KUKA KRL program: test.src

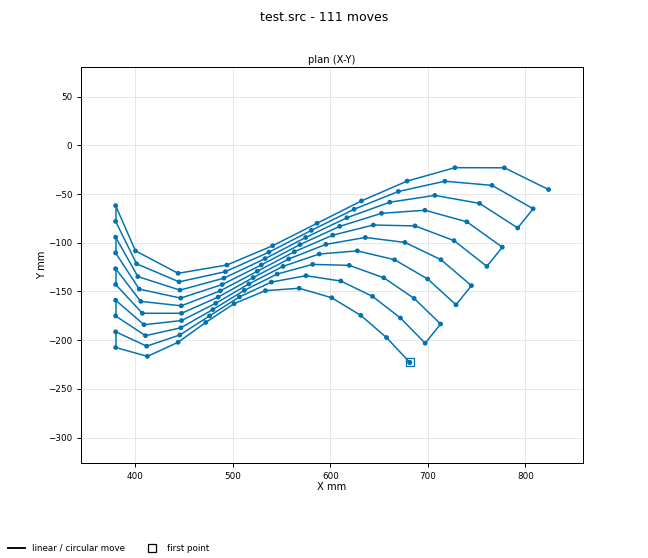
[picture p0: tool path of test.src, 111 of 113 moves have a stored position in this frame; points joined in program order, loops and branches not executed]
&ACCESS RVP
&REL 1
&PARAM TEMPLATE = C:\KRC\Roboter\Template\vorgabe
&PARAM EDITMASK = *
DEF test ( )


;FOLD INI
;FOLD BASISTECH INI
GLOBAL INTERRUPT DECL 3 WHEN $STOPMESS==TRUE DO IR_STOPM ( )
INTERRUPT ON 3
BAS (#INITMOV,0 )
;ENDFOLD (BASISTECH INI)
;ENDFOLD (INI)

;FOLD STARTPOSITION - BASE IS 0, TOOL IS 0, SPEED IS 15%, POSITION IS A1 5,A2 -90,A3 100,A4 5,A5 10,A6 -5,E1 0,E2 0,E3 0,E4 0
$BWDSTART = FALSE
PDAT_ACT = {VEL 15,ACC 100,APO_DIST 50}
FDAT_ACT = {TOOL_NO 0,BASE_NO 0,IPO_FRAME #BASE}
BAS (#PTP_PARAMS,15)
PTP  {A1 5,A2 -90,A3 100,A4 5,A5 10,A6 -5,E1 0,E2 0,E3 0,E4 0}
;ENDFOLD

;FOLD LIN SPEED IS 0.25 m/sec, INTERPOLATION SETTINGS IN FOLD
$VEL.CP=0.25
$APO.CDIS=10
$ADVANCE=3
;ENDFOLD

$OUT_C[1]=TRUE
PTP {E6POS: X 681.378, Y -222.764, Z 500, A 0, B -90, C 40.701, E1 0, E2 0, E3 0, E4 0, S 'B 110'} C_PTP
$VEL.CP=0.11208624
$OUT_C[1]=TRUE
LIN {E6POS: X 681.378, Y -222.764, Z 500, A 0, B -90, C 40.701, E1 0, E2 0, E3 0, E4 0} C_DIS
$VEL.CP=0.1175562
LIN {E6POS: X 657.556, Y -197.262, Z 500, A 0, B -90, C 45.729, E1 0, E2 0, E3 0, E4 0} C_DIS
$VEL.CP=0.12712281
LIN {E6POS: X 631.136, Y -174.483, Z 500, A 0, B -90, C 53.29, E1 0, E2 0, E3 0, E4 0} C_DIS
$VEL.CP=0.14338495
LIN {E6POS: X 601.341, Y -156.414, Z 500, A 0, B -90, C 65.177, E1 0, E2 0, E3 0, E4 0} C_DIS
$VEL.CP=0.16124801
LIN {E6POS: X 567.97, Y -146.683, Z 500, A 0, B -90, C 83.337, E1 0, E2 0, E3 0, E4 0} C_DIS
$VEL.CP=0.15591648
LIN {E6POS: X 533.344, Y -149.111, Z 500, A 0, B -90, C 104.356, E1 0, E2 0, E3 0, E4 0} C_DIS
$VEL.CP=0.13138869
LIN {E6POS: X 501.213, Y -162.493, Z 500, A 0, B -90, C 119.461, E1 0, E2 0, E3 0, E4 0} C_DIS
$VEL.CP=0.10713721
LIN {E6POS: X 472.106, Y -181.729, Z 500, A 0, B -90, C 126.091, E1 0, E2 0, E3 0, E4 0} C_DIS
$VEL.CP=0.12689649
LIN {E6POS: X 443.773, Y -202.115, Z 500, A 0, B -90, C 123.452, E1 0, E2 0, E3 0, E4 0} C_DIS
$VEL.CP=0.22954467
LIN {E6POS: X 412.246, Y -216.53, Z 500, A 0, B -90, C 99.792, E1 0, E2 0, E3 0, E4 0} C_DIS
$VEL.CP=0.19782427
LIN {E6POS: X 379.699, Y -207.447, Z 500, A 0, B -90, C 51.492, E1 0, E2 0, E3 0, E4 0} C_DIS
$VEL.CP=0.18350544
LIN {E6POS: X 379.699, Y -191.28, Z 500, A 0, B -90, C -136.662, E1 0, E2 0, E3 0, E4 0} C_DIS
$VEL.CP=0.242284
LIN {E6POS: X 411.548, Y -206.08, Z 500, A 0, B -90, C -88.625, E1 0, E2 0, E3 0, E4 0} C_DIS
$VEL.CP=0.13252691
LIN {E6POS: X 445.551, Y -194.567, Z 500, A 0, B -90, C -60.589, E1 0, E2 0, E3 0, E4 0} C_DIS
$VEL.CP=0.10130669
LIN {E6POS: X 476.069, Y -175.016, Z 500, A 0, B -90, C -56.087, E1 0, E2 0, E3 0, E4 0} C_DIS
$VEL.CP=0.12101501
LIN {E6POS: X 506.648, Y -155.559, Z 500, A 0, B -90, C -60.177, E1 0, E2 0, E3 0, E4 0} C_DIS
$VEL.CP=0.14114481
LIN {E6POS: X 539.479, Y -140.317, Z 500, A 0, B -90, C -71.221, E1 0, E2 0, E3 0, E4 0} C_DIS
$VEL.CP=0.15549513
LIN {E6POS: X 574.997, Y -133.814, Z 500, A 0, B -90, C -88.912, E1 0, E2 0, E3 0, E4 0} C_DIS
$VEL.CP=0.14877746
LIN {E6POS: X 610.665, Y -139.264, Z 500, A 0, B -90, C -108.055, E1 0, E2 0, E3 0, E4 0} C_DIS
$VEL.CP=0.13304864
LIN {E6POS: X 643.215, Y -155.004, Z 500, A 0, B -90, C -122.625, E1 0, E2 0, E3 0, E4 0} C_DIS
$VEL.CP=0.1215327
LIN {E6POS: X 671.847, Y -177.173, Z 500, A 0, B -90, C -132.204, E1 0, E2 0, E3 0, E4 0} C_DIS
$VEL.CP=0.11461978
LIN {E6POS: X 697.2, Y -203.06, Z 500, A 0, B -90, C -138.566, E1 0, E2 0, E3 0, E4 0} C_DIS
$VEL.CP=0.11747553
LIN {E6POS: X 713.022, Y -183.357, Z 500, A 0, B -90, C 42.204, E1 0, E2 0, E3 0, E4 0} C_DIS
$VEL.CP=0.12604367
LIN {E6POS: X 685.918, Y -157.123, Z 500, A 0, B -90, C 50.194, E1 0, E2 0, E3 0, E4 0} C_DIS
$VEL.CP=0.13895214
LIN {E6POS: X 654.762, Y -135.927, Z 500, A 0, B -90, C 62.153, E1 0, E2 0, E3 0, E4 0} C_DIS
$VEL.CP=0.15060037
LIN {E6POS: X 619.368, Y -123.2, Z 500, A 0, B -90, C 79.05, E1 0, E2 0, E3 0, E4 0} C_DIS
$VEL.CP=0.14631891
LIN {E6POS: X 581.798, Y -122.186, Z 500, A 0, B -90, C 97.587, E1 0, E2 0, E3 0, E4 0} C_DIS
$VEL.CP=0.12977299
LIN {E6POS: X 545.471, Y -132.089, Z 500, A 0, B -90, C 111.844, E1 0, E2 0, E3 0, E4 0} C_DIS
$VEL.CP=0.11350675
LIN {E6POS: X 511.672, Y -148.834, Z 500, A 0, B -90, C 119.873, E1 0, E2 0, E3 0, E4 0} C_DIS
$VEL.CP=0.1031691
LIN {E6POS: X 479.457, Y -168.509, Z 500, A 0, B -90, C 121.926, E1 0, E2 0, E3 0, E4 0} C_DIS
$VEL.CP=0.13868728
LIN {E6POS: X 446.677, Y -187.191, Z 500, A 0, B -90, C 115.335, E1 0, E2 0, E3 0, E4 0} C_DIS
$VEL.CP=0.24988499
LIN {E6POS: X 410.331, Y -195.313, Z 500, A 0, B -90, C 82.591, E1 0, E2 0, E3 0, E4 0} C_DIS
$VEL.CP=0.17049267
LIN {E6POS: X 379.699, Y -175.112, Z 500, A 0, B -90, C 36.664, E1 0, E2 0, E3 0, E4 0} C_DIS
$VEL.CP=0.15965107
LIN {E6POS: X 379.699, Y -158.945, Z 500, A 0, B -90, C -148.742, E1 0, E2 0, E3 0, E4 0} C_DIS
$VEL.CP=0.25
LIN {E6POS: X 408.793, Y -184.08, Z 500, A 0, B -90, C -106.079, E1 0, E2 0, E3 0, E4 0} C_DIS
$VEL.CP=0.14513617
LIN {E6POS: X 447.236, Y -179.828, Z 500, A 0, B -90, C -68.773, E1 0, E2 0, E3 0, E4 0} C_DIS
$VEL.CP=0.10734447
LIN {E6POS: X 482.361, Y -162.109, Z 500, A 0, B -90, C -60.049, E1 0, E2 0, E3 0, E4 0} C_DIS
$VEL.CP=0.10792353
LIN {E6POS: X 516.364, Y -142.247, Z 500, A 0, B -90, C -60.383, E1 0, E2 0, E3 0, E4 0} C_DIS
$VEL.CP=0.12129846
LIN {E6POS: X 551.369, Y -124.246, Z 500, A 0, B -90, C -66.049, E1 0, E2 0, E3 0, E4 0} C_DIS
$VEL.CP=0.13674186
LIN {E6POS: X 588.577, Y -111.545, Z 500, A 0, B -90, C -77.229, E1 0, E2 0, E3 0, E4 0} C_DIS
$VEL.CP=0.14833769
LIN {E6POS: X 627.681, Y -108.322, Z 500, A 0, B -90, C -94.073, E1 0, E2 0, E3 0, E4 0} C_DIS
$VEL.CP=0.14398834
LIN {E6POS: X 665.817, Y -117.427, Z 500, A 0, B -90, C -112.461, E1 0, E2 0, E3 0, E4 0} C_DIS
$VEL.CP=0.13105502
LIN {E6POS: X 699.766, Y -137.17, Z 500, A 0, B -90, C -127.03, E1 0, E2 0, E3 0, E4 0} C_DIS
$VEL.CP=0.12069929
LIN {E6POS: X 728.844, Y -163.654, Z 500, A 0, B -90, C -136.944, E1 0, E2 0, E3 0, E4 0} C_DIS
$VEL.CP=0.1243438
LIN {E6POS: X 744.665, Y -143.95, Z 500, A 0, B -90, C 43.947, E1 0, E2 0, E3 0, E4 0} C_DIS
$VEL.CP=0.13643728
LIN {E6POS: X 713.389, Y -117.376, Z 500, A 0, B -90, C 56.167, E1 0, E2 0, E3 0, E4 0} C_DIS
$VEL.CP=0.14714289
LIN {E6POS: X 676.456, Y -99.656, Z 500, A 0, B -90, C 73.323, E1 0, E2 0, E3 0, E4 0} C_DIS
$VEL.CP=0.14302107
LIN {E6POS: X 635.84, Y -94.578, Z 500, A 0, B -90, C 92.121, E1 0, E2 0, E3 0, E4 0} C_DIS
$VEL.CP=0.12834552
LIN {E6POS: X 595.443, Y -101.629, Z 500, A 0, B -90, C 106.677, E1 0, E2 0, E3 0, E4 0} C_DIS
$VEL.CP=0.11500083
LIN {E6POS: X 557.21, Y -116.656, Z 500, A 0, B -90, C 115.335, E1 0, E2 0, E3 0, E4 0} C_DIS
$VEL.CP=0.10366841
LIN {E6POS: X 520.795, Y -135.736, Z 500, A 0, B -90, C 119.205, E1 0, E2 0, E3 0, E4 0} C_DIS
$VEL.CP=0.11093951
LIN {E6POS: X 484.87, Y -155.738, Z 500, A 0, B -90, C 118.025, E1 0, E2 0, E3 0, E4 0} C_DIS
$VEL.CP=0.15165687
LIN {E6POS: X 447.326, Y -172.357, Z 500, A 0, B -90, C 107.094, E1 0, E2 0, E3 0, E4 0} C_DIS
$VEL.CP=0.24285384
LIN {E6POS: X 407.124, Y -172.341, Z 500, A 0, B -90, C 65.741, E1 0, E2 0, E3 0, E4 0} C_DIS
$VEL.CP=0.15093802
LIN {E6POS: X 379.699, Y -142.777, Z 500, A 0, B -90, C 26.821, E1 0, E2 0, E3 0, E4 0} C_DIS
$VEL.CP=0.14400658
LIN {E6POS: X 379.699, Y -126.61, Z 500, A 0, B -90, C -156.794, E1 0, E2 0, E3 0, E4 0} C_DIS
$VEL.CP=0.23087273
LIN {E6POS: X 405.466, Y -160.137, Z 500, A 0, B -90, C -121.592, E1 0, E2 0, E3 0, E4 0} C_DIS
$VEL.CP=0.15801723
LIN {E6POS: X 447.042, Y -164.693, Z 500, A 0, B -90, C -77.117, E1 0, E2 0, E3 0, E4 0} C_DIS
$VEL.CP=0.11407162
LIN {E6POS: X 487.06, Y -149.339, Z 500, A 0, B -90, C -63.896, E1 0, E2 0, E3 0, E4 0} C_DIS
$VEL.CP=0.10035442
LIN {E6POS: X 525.025, Y -129.253, Z 500, A 0, B -90, C -61.385, E1 0, E2 0, E3 0, E4 0} C_DIS
$VEL.CP=0.1102753
LIN {E6POS: X 563.021, Y -109.226, Z 500, A 0, B -90, C -63.717, E1 0, E2 0, E3 0, E4 0} C_DIS
$VEL.CP=0.12153792
LIN {E6POS: X 602.44, Y -92.222, Z 500, A 0, B -90, C -70.369, E1 0, E2 0, E3 0, E4 0} C_DIS
$VEL.CP=0.136359
LIN {E6POS: X 644.03, Y -81.81, Z 500, A 0, B -90, C -82.534, E1 0, E2 0, E3 0, E4 0} C_DIS
$VEL.CP=0.14766606
LIN {E6POS: X 686.794, Y -82.719, Z 500, A 0, B -90, C -100.715, E1 0, E2 0, E3 0, E4 0} C_DIS
$VEL.CP=0.14192006
LIN {E6POS: X 726.787, Y -97.808, Z 500, A 0, B -90, C -120.207, E1 0, E2 0, E3 0, E4 0} C_DIS
$VEL.CP=0.12846969
LIN {E6POS: X 760.487, Y -124.247, Z 500, A 0, B -90, C -135.081, E1 0, E2 0, E3 0, E4 0} C_DIS
$VEL.CP=0.13314639
LIN {E6POS: X 776.309, Y -104.544, Z 500, A 0, B -90, C 45.972, E1 0, E2 0, E3 0, E4 0} C_DIS
$VEL.CP=0.14706142
LIN {E6POS: X 739.968, Y -78.534, Z 500, A 0, B -90, C 63.896, E1 0, E2 0, E3 0, E4 0} C_DIS
$VEL.CP=0.14550026
LIN {E6POS: X 696.968, Y -66.648, Z 500, A 0, B -90, C 85.122, E1 0, E2 0, E3 0, E4 0} C_DIS
$VEL.CP=0.12971982
LIN {E6POS: X 652.368, Y -69.816, Z 500, A 0, B -90, C 101.827, E1 0, E2 0, E3 0, E4 0} C_DIS
$VEL.CP=0.11619168
LIN {E6POS: X 609.584, Y -83.16, Z 500, A 0, B -90, C 111.844, E1 0, E2 0, E3 0, E4 0} C_DIS
$VEL.CP=0.10667887
LIN {E6POS: X 568.822, Y -101.888, Z 500, A 0, B -90, C 116.873, E1 0, E2 0, E3 0, E4 0} C_DIS
$VEL.CP=0.10183953
LIN {E6POS: X 529.103, Y -122.765, Z 500, A 0, B -90, C 117.975, E1 0, E2 0, E3 0, E4 0} C_DIS
$VEL.CP=0.1168252
LIN {E6POS: X 488.996, Y -142.872, Z 500, A 0, B -90, C 114.207, E1 0, E2 0, E3 0, E4 0} C_DIS
$VEL.CP=0.16396278
LIN {E6POS: X 446.474, Y -156.78, Z 500, A 0, B -90, C 98.681, E1 0, E2 0, E3 0, E4 0} C_DIS
$VEL.CP=0.21696831
LIN {E6POS: X 403.904, Y -147.552, Z 500, A 0, B -90, C 51.984, E1 0, E2 0, E3 0, E4 0} C_DIS
$VEL.CP=0.13847707
LIN {E6POS: X 379.699, Y -110.442, Z 500, A 0, B -90, C 20.174, E1 0, E2 0, E3 0, E4 0} C_DIS
$VEL.CP=0.13402625
LIN {E6POS: X 379.699, Y -94.275, Z 500, A 0, B -90, C -162.362, E1 0, E2 0, E3 0, E4 0} C_DIS
$VEL.CP=0.20326516
LIN {E6POS: X 402.478, Y -134.673, Z 500, A 0, B -90, C -133.461, E1 0, E2 0, E3 0, E4 0} C_DIS
$VEL.CP=0.16923532
LIN {E6POS: X 445.699, Y -148.587, Z 500, A 0, B -90, C -85.584, E1 0, E2 0, E3 0, E4 0} C_DIS
$VEL.CP=0.11925948
LIN {E6POS: X 490.735, Y -136.312, Z 500, A 0, B -90, C -67.667, E1 0, E2 0, E3 0, E4 0} C_DIS
$VEL.CP=0.10395698
LIN {E6POS: X 533.068, Y -116.245, Z 500, A 0, B -90, C -62.743, E1 0, E2 0, E3 0, E4 0} C_DIS
$VEL.CP=0.1039008
LIN {E6POS: X 574.631, Y -94.594, Z 500, A 0, B -90, C -62.82, E1 0, E2 0, E3 0, E4 0} C_DIS
$VEL.CP=0.11203091
LIN {E6POS: X 616.876, Y -74.326, Z 500, A 0, B -90, C -66.538, E1 0, E2 0, E3 0, E4 0} C_DIS
$VEL.CP=0.12381166
LIN {E6POS: X 660.911, Y -58.406, Z 500, A 0, B -90, C -74.629, E1 0, E2 0, E3 0, E4 0} C_DIS
$VEL.CP=0.1413023
LIN {E6POS: X 707.115, Y -51.403, Z 500, A 0, B -90, C -89.484, E1 0, E2 0, E3 0, E4 0} C_DIS
$VEL.CP=0.15127063
LIN {E6POS: X 752.951, Y -59.624, Z 500, A 0, B -90, C -111.663, E1 0, E2 0, E3 0, E4 0} C_DIS
$VEL.CP=0.138453
LIN {E6POS: X 792.131, Y -84.84, Z 500, A 0, B -90, C -132.852, E1 0, E2 0, E3 0, E4 0} C_DIS
$VEL.CP=0.14447882
LIN {E6POS: X 807.953, Y -65.137, Z 500, A 0, B -90, C 48.405, E1 0, E2 0, E3 0, E4 0} C_DIS
$VEL.CP=0.15392265
LIN {E6POS: X 765.772, Y -41.137, Z 500, A 0, B -90, C 73.142, E1 0, E2 0, E3 0, E4 0} C_DIS
$VEL.CP=0.13604527
LIN {E6POS: X 717.348, Y -36.888, Z 500, A 0, B -90, C 95.334, E1 0, E2 0, E3 0, E4 0} C_DIS
$VEL.CP=0.11884865
LIN {E6POS: X 669.682, Y -47.421, Z 500, A 0, B -90, C 108.236, E1 0, E2 0, E3 0, E4 0} C_DIS
$VEL.CP=0.10878646
LIN {E6POS: X 624.311, Y -65.639, Z 500, A 0, B -90, C 114.719, E1 0, E2 0, E3 0, E4 0} C_DIS
$VEL.CP=0.10172496
LIN {E6POS: X 580.461, Y -87.313, Z 500, A 0, B -90, C 117.308, E1 0, E2 0, E3 0, E4 0} C_DIS
$VEL.CP=0.10568283
LIN {E6POS: X 536.955, Y -109.677, Z 500, A 0, B -90, C 116.488, E1 0, E2 0, E3 0, E4 0} C_DIS
$VEL.CP=0.12141577
LIN {E6POS: X 492.32, Y -129.643, Z 500, A 0, B -90, C 110.482, E1 0, E2 0, E3 0, E4 0} C_DIS
$VEL.CP=0.17360632
LIN {E6POS: X 444.786, Y -140.103, Z 500, A 0, B -90, C 90.229, E1 0, E2 0, E3 0, E4 0} C_DIS
$VEL.CP=0.19085942
LIN {E6POS: X 401.196, Y -121.577, Z 500, A 0, B -90, C 41.962, E1 0, E2 0, E3 0, E4 0} C_DIS
$VEL.CP=0.13040204
LIN {E6POS: X 379.699, Y -78.107, Z 500, A 0, B -90, C 15.481, E1 0, E2 0, E3 0, E4 0} C_DIS
$VEL.CP=0.12741441
LIN {E6POS: X 379.699, Y -61.94, Z 500, A 0, B -90, C -166.353, E1 0, E2 0, E3 0, E4 0} C_DIS
$VEL.CP=0.18011377
LIN {E6POS: X 400.051, Y -108.327, Z 500, A 0, B -90, C -141.904, E1 0, E2 0, E3 0, E4 0} C_DIS
$VEL.CP=0.17691218
LIN {E6POS: X 443.794, Y -131.331, Z 500, A 0, B -90, C -93.841, E1 0, E2 0, E3 0, E4 0} C_DIS
$VEL.CP=0.12332322
LIN {E6POS: X 493.791, Y -122.855, Z 500, A 0, B -90, C -71.329, E1 0, E2 0, E3 0, E4 0} C_DIS
$VEL.CP=0.10710207
LIN {E6POS: X 540.788, Y -103.051, Z 500, A 0, B -90, C -64.28, E1 0, E2 0, E3 0, E4 0} C_DIS
$VEL.CP=0.1
LIN {E6POS: X 586.324, Y -80.022, Z 500, A 0, B -90, C -62.666, E1 0, E2 0, E3 0, E4 0} C_DIS
$VEL.CP=0.10623915
LIN {E6POS: X 631.885, Y -57.04, Z 500, A 0, B -90, C -64.332, E1 0, E2 0, E3 0, E4 0} C_DIS
$VEL.CP=0.11479347
LIN {E6POS: X 678.684, Y -36.738, Z 500, A 0, B -90, C -69.518, E1 0, E2 0, E3 0, E4 0} C_DIS
$VEL.CP=0.13058396
LIN {E6POS: X 727.745, Y -22.981, Z 500, A 0, B -90, C -80.5, E1 0, E2 0, E3 0, E4 0} C_DIS
$VEL.CP=0.15455497
LIN {E6POS: X 778.478, Y -23.118, Z 500, A 0, B -90, C -101.883, E1 0, E2 0, E3 0, E4 0} C_DIS
$VEL.CP=0.15132345
LIN {E6POS: X 823.775, Y -45.434, Z 500, A 0, B -90, C -130.253, E1 0, E2 0, E3 0, E4 0} C_DIS
$OUT_C[1]=FALSE
PTP {E6AXIS: A1 5, A2 -90, A3 100, A4 5, A5 10, A6 -5, E1 0, E2 0, E3 0, E4 0} C_PTP

END
